FUNCTION_BLOCK DirectOnlineStarterMotor implements I_SingleDirectionMotor
VAR
	contactor	:	Contactor;
END_VAR

METHOD PUBLIC Start
VAR_INPUT
END_VAR
contactor.SwitchOn();
END_METHOD

METHOD PUBLIC Stop
VAR_INPUT
END_VAR
contactor.SwitchOff();
END_METHOD

END_FUNCTION_BLOCK

(* stored: Version 1.1.0.1, ProductVersion 3.1.4024.11
   POU DirectOnlineStarterMotor: Id {d1e95a37-c50a-4020-8ecb-f6b8ea091542}, SpecialFunc None
   Method Start: Id {584e866d-7b71-4da9-8644-e945068d53e4}
   Method Stop: Id {92ae5ef7-1491-4250-9599-f019de641b56} *)
